// TIA Portal V19 export
VAR_GLOBAL   // PLC tag table "D20"
   D20_Lp_EntryReq_LB302 AT %Q200.7 : Bool;   // 260SH1
   D20_Lp_SafetyReset_LB302 AT %Q201.0 : Bool;   // 260SH2
   D20_Pb_EntryReq_LB302 AT %I201.0 : Bool;   // 260SH1
   D20_Pb_SafetyReset_LB302 AT %I201.1 : Bool;   // 260SH2
   D20_Comando_Elettroserratura AT %Q200.6 : Bool;   // 26202
   D20_Cancello_Chiuso AT %I200.6 : Bool;   // 26201
   D20_Cancello_Bloccato AT %I200.7 : Bool;   // 26003
   D20_Ls_Os1 AT %I1200.3 : Bool;   // 200DI3 - 260A1
   D20_Ls_Os2 AT %I1200.7 : Bool;   // 200DI7 - 260A1
END_VAR
